{attribute 'qualified_only'}
VAR_GLOBAL
	//cycle times
	tTaskCycleTime_MAIN				: TIME := T#10MS;
	tCtrlCycleTime_MAIN				: TIME := T#5S;
END_VAR

(* stored: Version 1.1.0.1, ProductVersion 3.1.4024.6
   GVL GlobalVariables: Id {8a6aab08-6efe-48c3-a056-92271920ea20} *)
